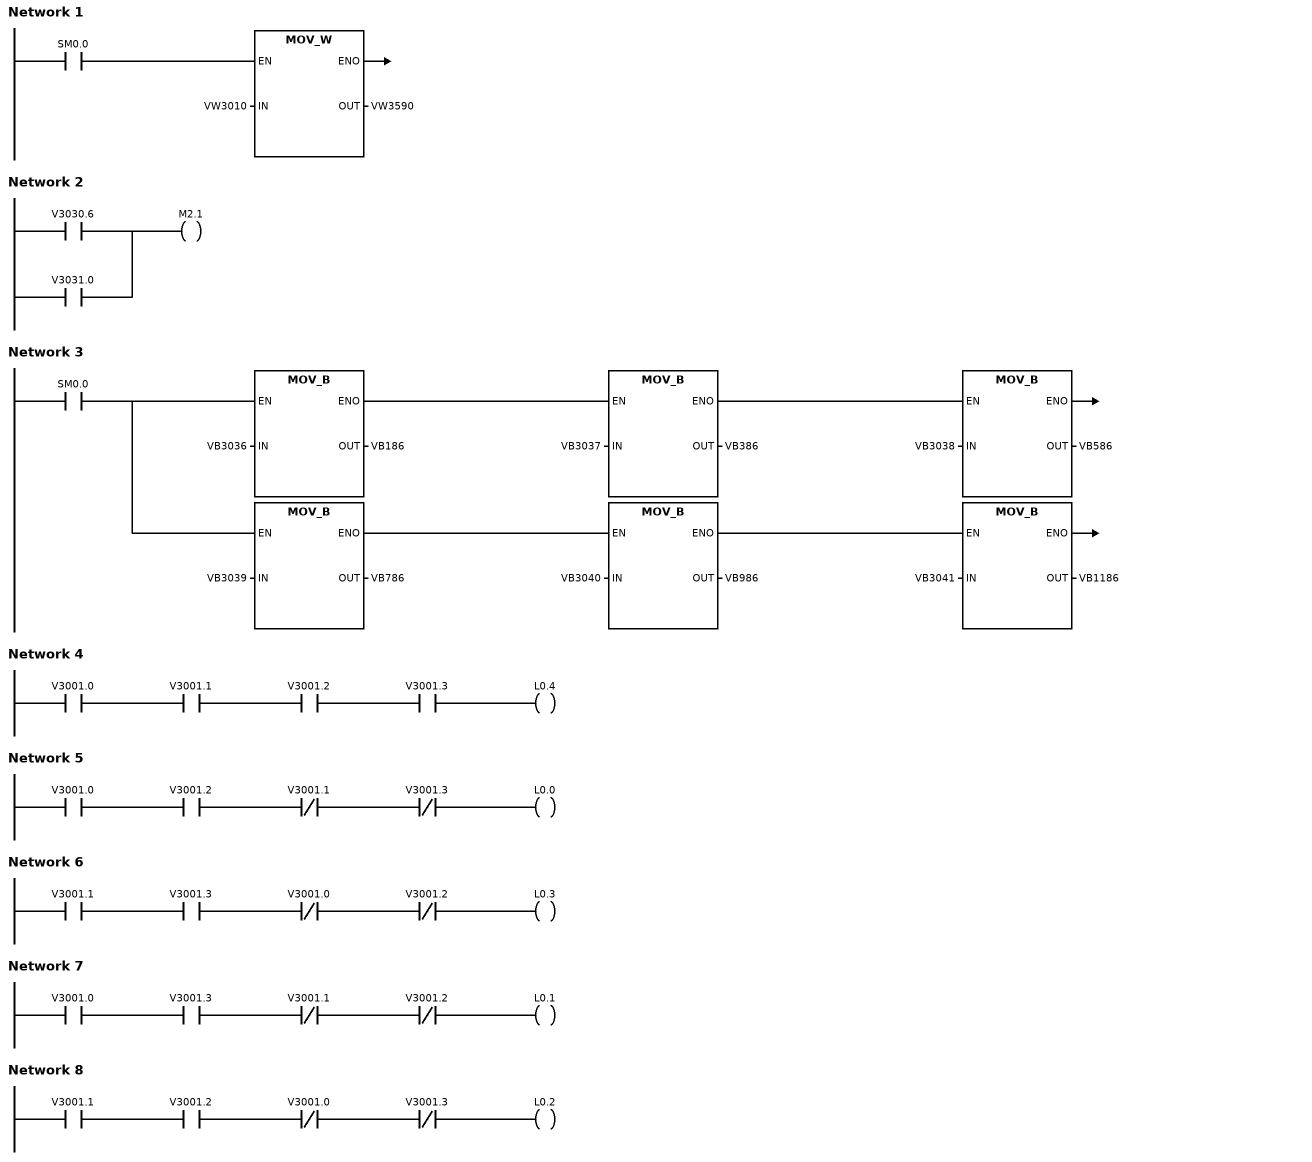
[picture p72: SBR10 networks 1-8]
Network 1
LD     SM0.0
MOVW   VW3010, VW3590
Network 2
LD     V3030.6
O      V3031.0
=      M2.1
Network 3
LD     SM0.0
LPS
MOVB   VB3036, VB186
AENO
MOVB   VB3037, VB386
AENO
MOVB   VB3038, VB586
LPP
MOVB   VB3039, VB786
AENO
MOVB   VB3040, VB986
AENO
MOVB   VB3041, VB1186
Network 4
LD     V3001.0
A      V3001.1
A      V3001.2
A      V3001.3
=      L0.4
Network 5
LD     V3001.0
A      V3001.2
AN     V3001.1
AN     V3001.3
=      L0.0
Network 6
LD     V3001.1
A      V3001.3
AN     V3001.0
AN     V3001.2
=      L0.3
Network 7
LD     V3001.0
A      V3001.3
AN     V3001.1
AN     V3001.2
=      L0.1
Network 8
LD     V3001.1
A      V3001.2
AN     V3001.0
AN     V3001.3
=      L0.2
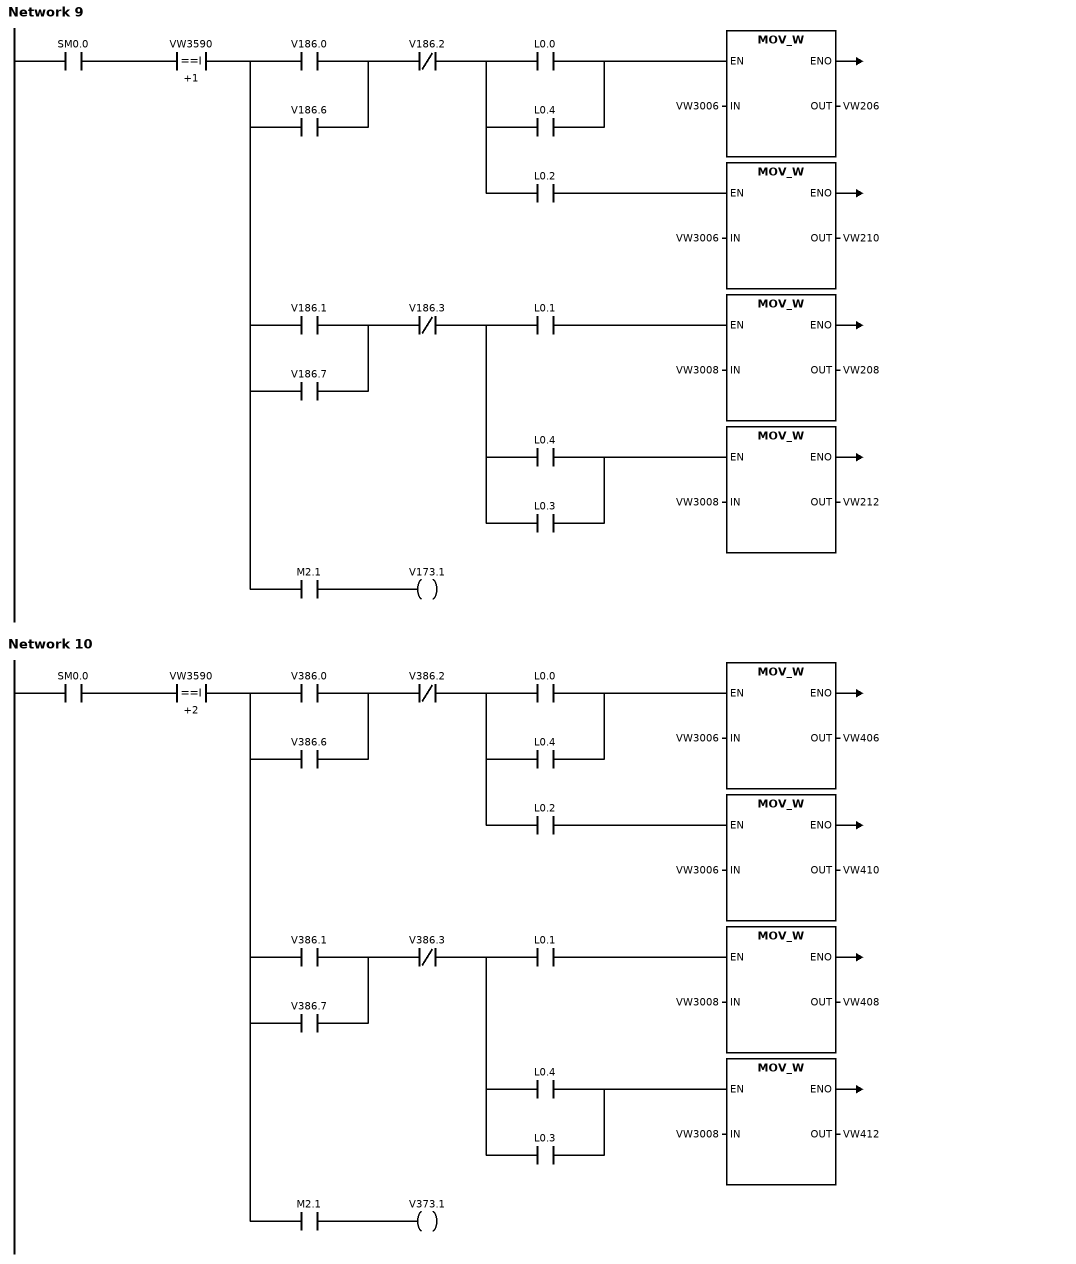
Network 9
LD     SM0.0
AW=    VW3590, +1
LPS
LD     V186.0
O      V186.6
AN     V186.2
ALD
LPS
LD     L0.0
O      L0.4
ALD
MOVW   VW3006, VW206
LPP
A      L0.2
MOVW   VW3006, VW210
LRD
LD     V186.1
O      V186.7
AN     V186.3
ALD
LPS
A      L0.1
MOVW   VW3008, VW208
LPP
LD     L0.4
O      L0.3
ALD
MOVW   VW3008, VW212
LPP
A      M2.1
=      V173.1
Network 10
LD     SM0.0
AW=    VW3590, +2
LPS
LD     V386.0
O      V386.6
AN     V386.2
ALD
LPS
LD     L0.0
O      L0.4
ALD
MOVW   VW3006, VW406
LPP
A      L0.2
MOVW   VW3006, VW410
LRD
LD     V386.1
O      V386.7
AN     V386.3
ALD
LPS
A      L0.1
MOVW   VW3008, VW408
LPP
LD     L0.4
O      L0.3
ALD
MOVW   VW3008, VW412
LPP
A      M2.1
=      V373.1
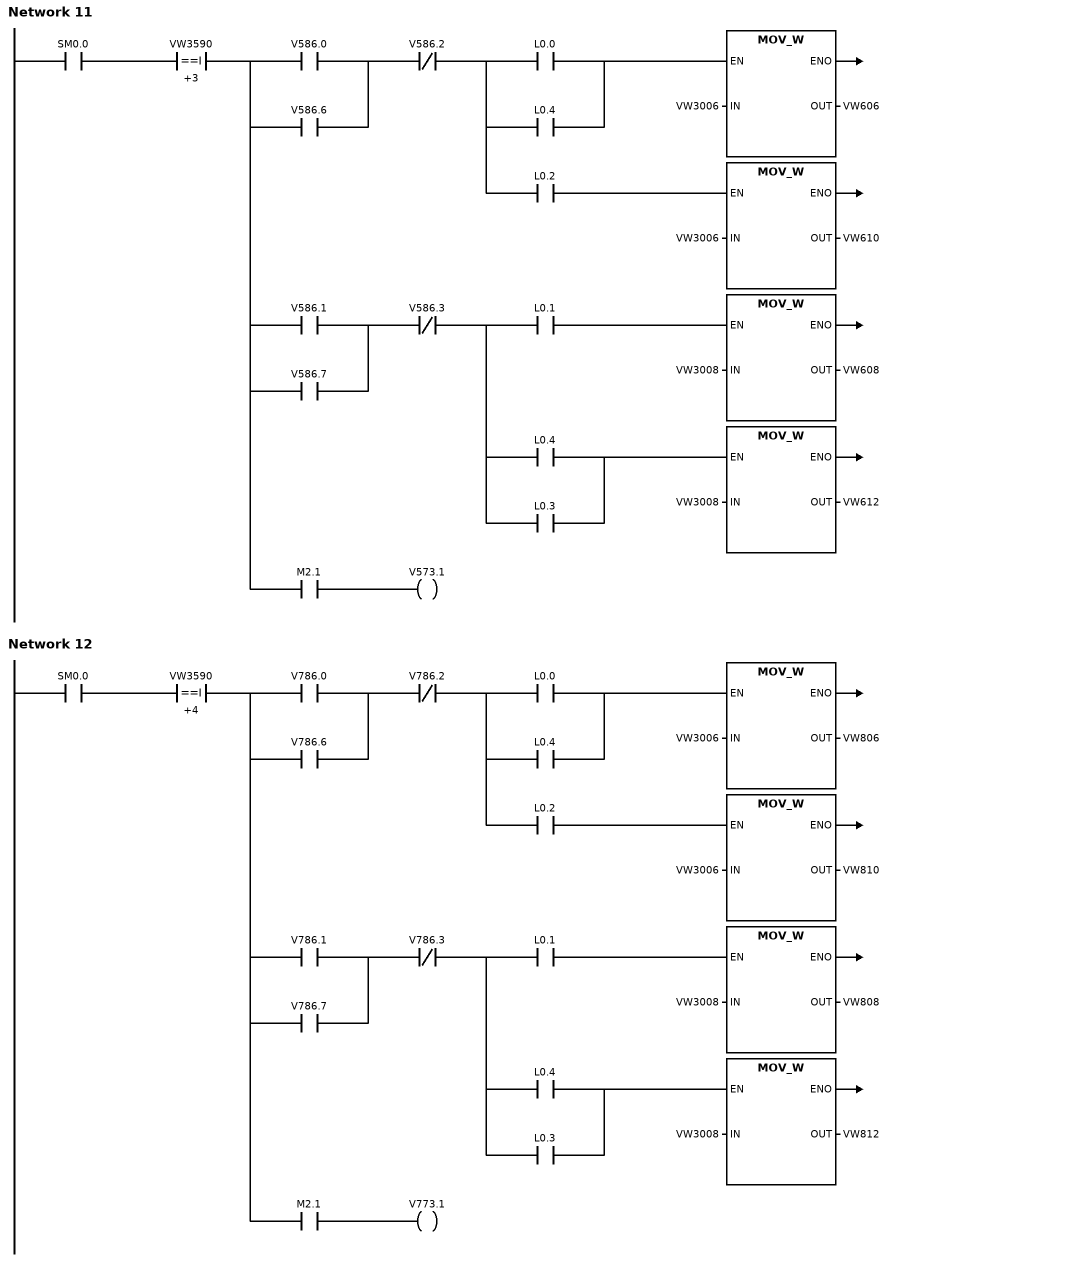
Network 11
LD     SM0.0
AW=    VW3590, +3
LPS
LD     V586.0
O      V586.6
AN     V586.2
ALD
LPS
LD     L0.0
O      L0.4
ALD
MOVW   VW3006, VW606
LPP
A      L0.2
MOVW   VW3006, VW610
LRD
LD     V586.1
O      V586.7
AN     V586.3
ALD
LPS
A      L0.1
MOVW   VW3008, VW608
LPP
LD     L0.4
O      L0.3
ALD
MOVW   VW3008, VW612
LPP
A      M2.1
=      V573.1
Network 12
LD     SM0.0
AW=    VW3590, +4
LPS
LD     V786.0
O      V786.6
AN     V786.2
ALD
LPS
LD     L0.0
O      L0.4
ALD
MOVW   VW3006, VW806
LPP
A      L0.2
MOVW   VW3006, VW810
LRD
LD     V786.1
O      V786.7
AN     V786.3
ALD
LPS
A      L0.1
MOVW   VW3008, VW808
LPP
LD     L0.4
O      L0.3
ALD
MOVW   VW3008, VW812
LPP
A      M2.1
=      V773.1
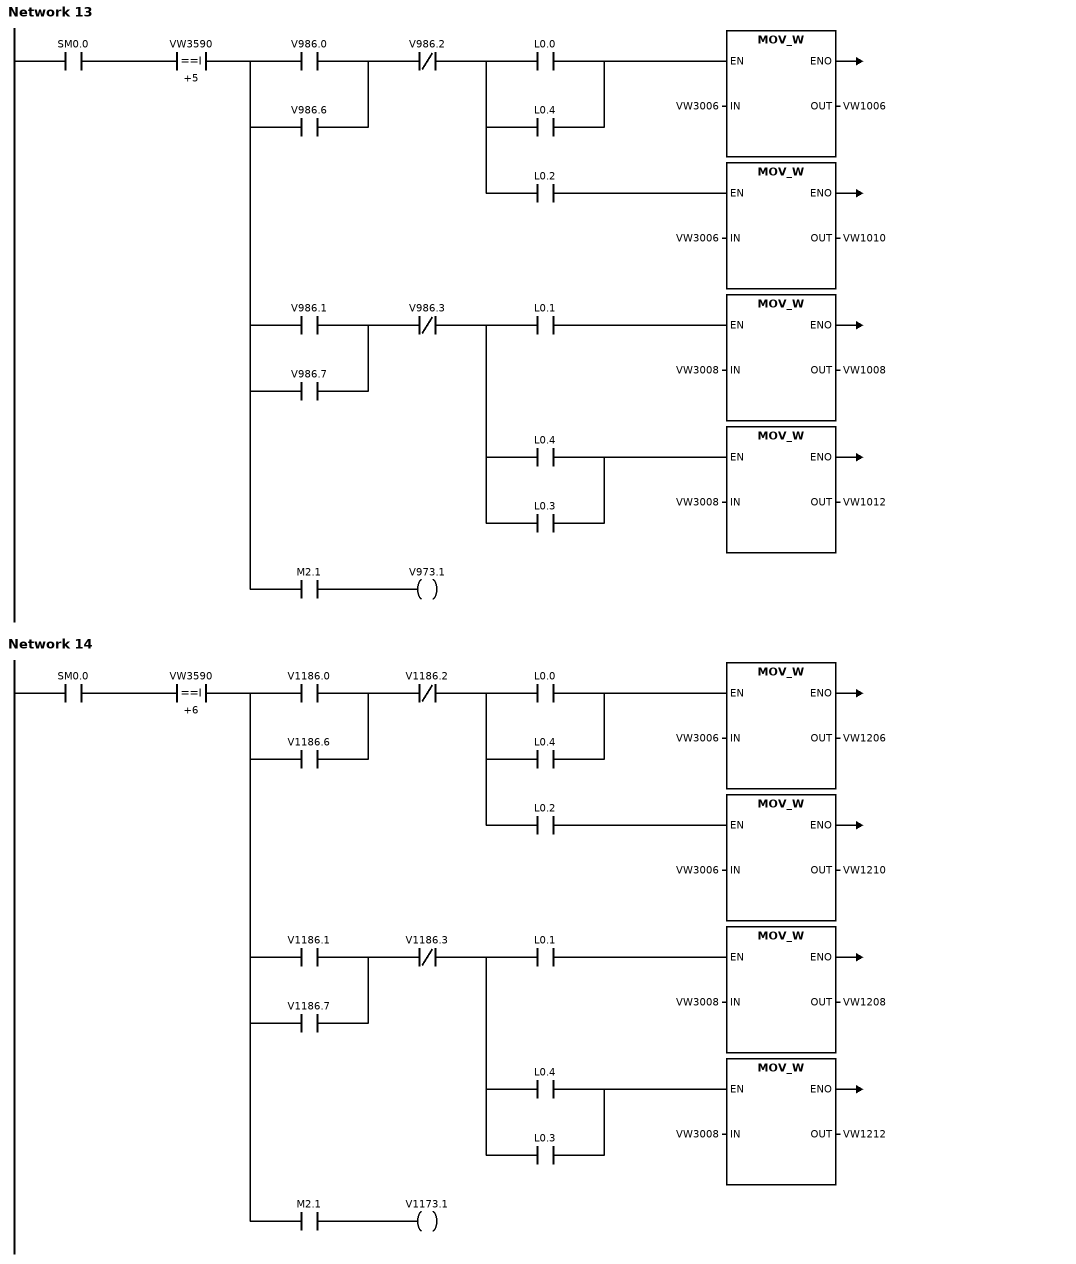
Network 13
LD     SM0.0
AW=    VW3590, +5
LPS
LD     V986.0
O      V986.6
AN     V986.2
ALD
LPS
LD     L0.0
O      L0.4
ALD
MOVW   VW3006, VW1006
LPP
A      L0.2
MOVW   VW3006, VW1010
LRD
LD     V986.1
O      V986.7
AN     V986.3
ALD
LPS
A      L0.1
MOVW   VW3008, VW1008
LPP
LD     L0.4
O      L0.3
ALD
MOVW   VW3008, VW1012
LPP
A      M2.1
=      V973.1
Network 14
LD     SM0.0
AW=    VW3590, +6
LPS
LD     V1186.0
O      V1186.6
AN     V1186.2
ALD
LPS
LD     L0.0
O      L0.4
ALD
MOVW   VW3006, VW1206
LPP
A      L0.2
MOVW   VW3006, VW1210
LRD
LD     V1186.1
O      V1186.7
AN     V1186.3
ALD
LPS
A      L0.1
MOVW   VW3008, VW1208
LPP
LD     L0.4
O      L0.3
ALD
MOVW   VW3008, VW1212
LPP
A      M2.1
=      V1173.1
END_SUBROUTINE_BLOCK

SUBROUTINE_BLOCK alarm_process:SBR11
TITLE=
BEGIN
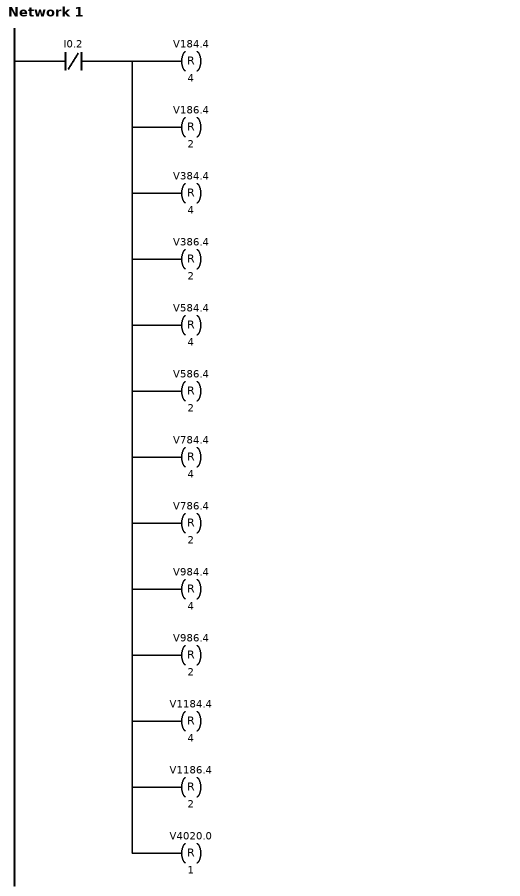
Network 1
LDN    I0.2
R      V184.4, 4
R      V186.4, 2
R      V384.4, 4
R      V386.4, 2
R      V584.4, 4
R      V586.4, 2
R      V784.4, 4
R      V786.4, 2
R      V984.4, 4
R      V986.4, 2
R      V1184.4, 4
R      V1186.4, 2
R      V4020.0, 1
END_SUBROUTINE_BLOCK

// SBR12: protected block, not included

SUBROUTINE_BLOCK auto_stop:SBR13
TITLE=
BEGIN
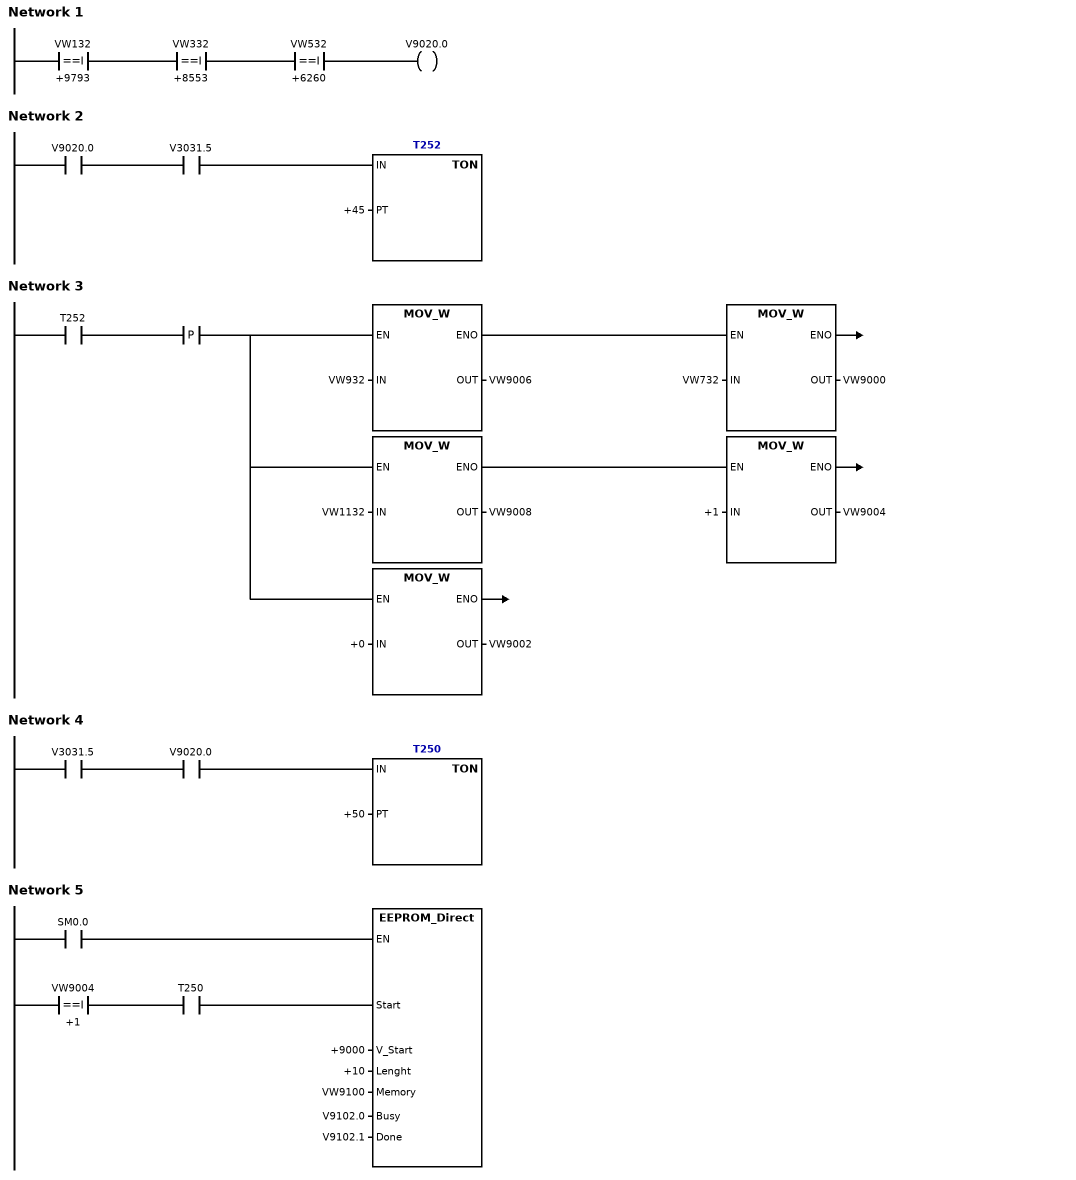
Network 1
LDW=   VW132, +9793
AW=    VW332, +8553
AW=    VW532, +6260
=      V9020.0
Network 2
LD     V9020.0
A      V3031.5
TON    T252, +45
Network 3
LD     T252
EU
LPS
MOVW   VW932, VW9006
AENO
MOVW   VW732, VW9000
LRD
MOVW   VW1132, VW9008
AENO
MOVW   +1, VW9004
LPP
MOVW   +0, VW9002
Network 4
LD     V3031.5
A      V9020.0
TON    T250, +50
Network 5
LD     SM0.0
=      L60.0
LDW=   VW9004, +1
A      T250
=      L63.7
LD     L60.0
CALL   EEPROM_Direct:SBR14, L63.7, +9000, +10, VW9100, V9102.0, V9102.1
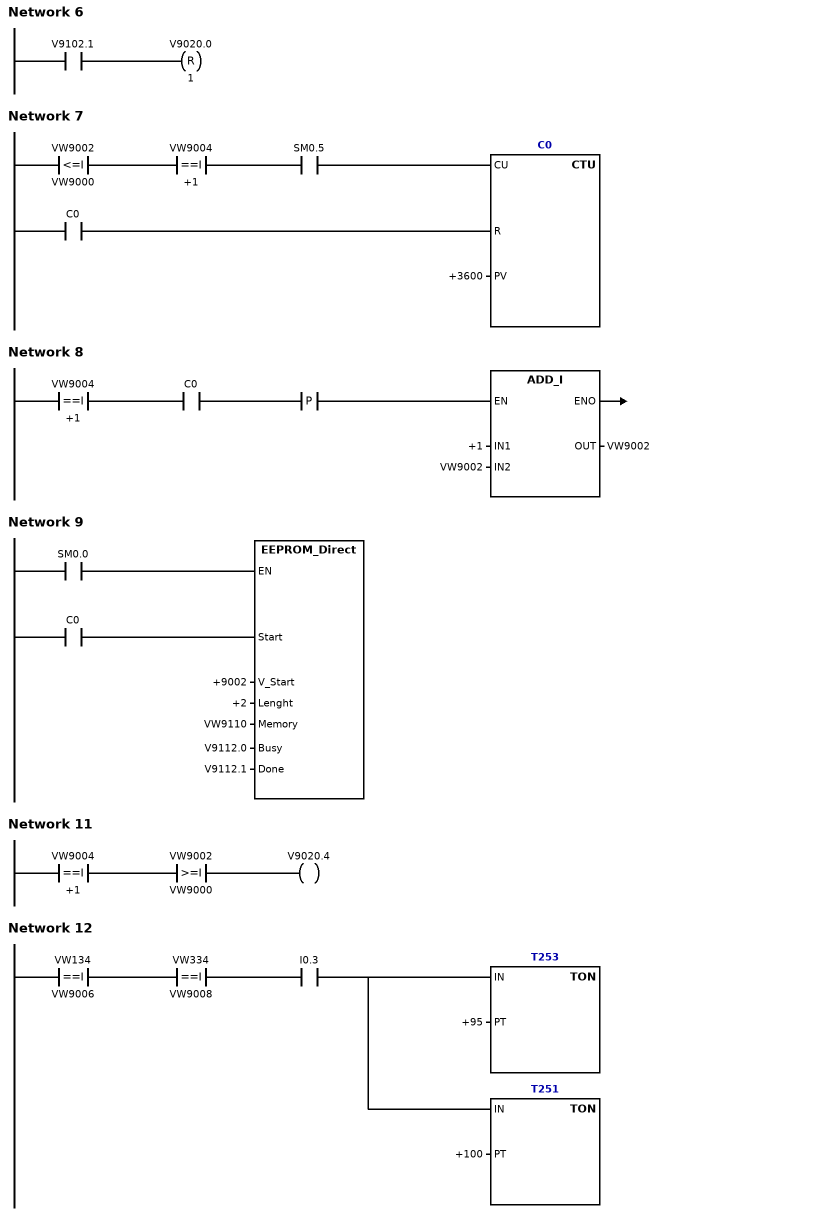
Network 6
LD     V9102.1
R      V9020.0, 1
Network 7
LDW<=  VW9002, VW9000
AW=    VW9004, +1
A      SM0.5
LD     C0
CTU    C0, +3600
Network 8
LDW=   VW9004, +1
A      C0
EU
+I     +1, VW9002
Network 9
LD     SM0.0
=      L60.0
LD     C0
=      L63.7
LD     L60.0
CALL   EEPROM_Direct:SBR14, L63.7, +9002, +2, VW9110, V9112.0, V9112.1
Network 11
LDW=   VW9004, +1
AW>=   VW9002, VW9000
=      V9020.4
Network 12
LDW=   VW134, VW9006
AW=    VW334, VW9008
A      I0.3
TON    T253, +95
TON    T251, +100
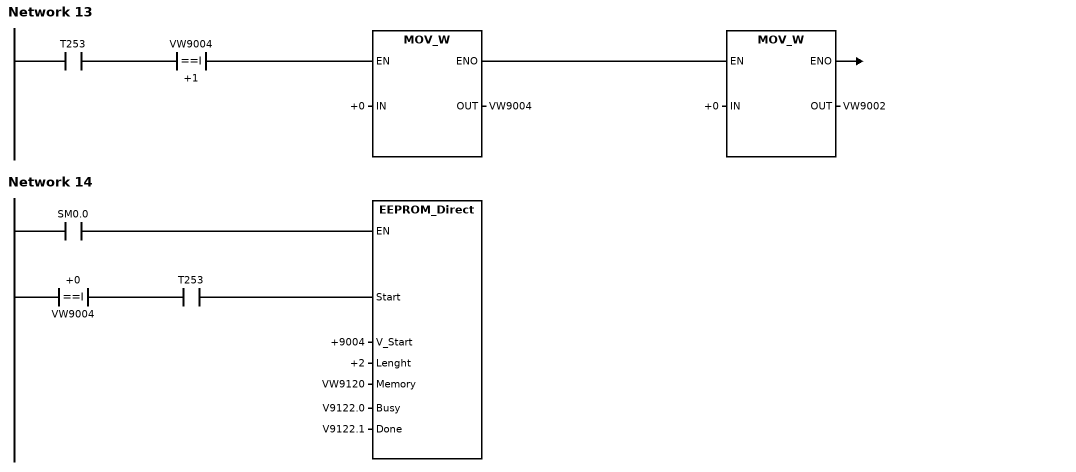
Network 13
LD     T253
AW=    VW9004, +1
MOVW   +0, VW9004
AENO
MOVW   +0, VW9002
Network 14
LD     SM0.0
=      L60.0
LDW=   +0, VW9004
A      T253
=      L63.7
LD     L60.0
CALL   EEPROM_Direct:SBR14, L63.7, +9004, +2, VW9120, V9122.0, V9122.1
END_SUBROUTINE_BLOCK

// SBR14: protected block, not included

// (further data pages could not be read)
